{attribute addProperty BoxType "EL1502--0000"}
{attribute addProperty Id "Enable_output_functionsAT %Q*BOOL811Set_outputAT %Q*BOOL812Set_counterAT %Q*BOOL813Inhibit_counterAT %Q*BOOL814Set_counter_valueAT %Q*UDINT32417"}
{attribute addProperty CRC "1515237018"}
{attribute addProperty SizeInBites "64"}
{attribute addProperty SizeInBytes "8"}
TYPE CNT_Outputs_5A50AE9A :
STRUCT
	{attribute addProperty Name "Enable_output_functions"}
	Enable_output_functions AT %Q* : BOOL;
	{attribute addProperty Name "Set_output"}
	Set_output AT %Q* : BOOL;
	{attribute addProperty Name "Set_counter"}
	Set_counter AT %Q* : BOOL;
	{attribute addProperty Name "Inhibit_counter"}
	Inhibit_counter AT %Q* : BOOL;
	{attribute addProperty Name "Set_counter_value"}
	Set_counter_value AT %Q* : UDINT;
END_STRUCT
END_TYPE

(* stored: Version 1.2.0.0, ProductVersion 3.1.4024.9
   DUT CNT_Outputs_5A50AE9A: Id {77c63c18-2821-4481-9d36-1789a429dba1} *)
